INTERFACE I_Inverter

PROPERTY ActualSpeed : REAL
GET
END_GET
END_PROPERTY

PROPERTY bIsMove : BOOL
GET
END_GET
END_PROPERTY

PROPERTY fTargetSpeed : REAL
GET
END_GET
SET
END_SET
END_PROPERTY

METHOD Reset : BOOL
VAR_INPUT
END_VAR
END_METHOD

METHOD Reverse : BOOL
VAR_INPUT
END_VAR
END_METHOD

METHOD Start : BOOL
VAR_INPUT
END_VAR
END_METHOD

METHOD Stop : BOOL
VAR_INPUT
END_VAR
END_METHOD

END_INTERFACE

(* stored: Version 1.1.0.1, ProductVersion 3.1.4024.12
   Itf I_Inverter: Id {711f4871-830e-4f42-bbe7-312b12f12c0a}
   Property ActualSpeed: Id {6b5b5053-377a-439e-972f-55220ffdb6f5}
   Get Get: Id {0a2198f7-ad7c-4d44-bef6-b6b1efa2a460}
   Property bIsMove: Id {423ff018-b570-43fb-92c2-a73a6f6aea59}
   Get Get: Id {a0160f4e-2cd8-4808-8615-6c03659a2eb7}
   Property fTargetSpeed: Id {b253edd2-271a-48b7-956e-e441ec9c010f}
   Get Get: Id {242c04aa-a6b1-4ab3-9553-ac653ceb0d80}
   Set Set: Id {63f34068-ab7e-4d84-ac8a-0aa642d38642}
   Method Reset: Id {1aefdc0a-91ff-4d60-845d-126182e6438d}
   Method Reverse: Id {d73a2ad3-2974-4cfd-b416-64234b544bd8}
   Method Start: Id {de90ca9b-6b89-46c5-a0a6-54da42b4611c}
   Method Stop: Id {cce98897-420f-4d8a-a556-74aa88c6b77d} *)
